{attribute 'call_after_init'}
FUNCTION_BLOCK FB_eVWithinSpec_Test EXTENDS TcUnit.FB_TestSuite
VAR_INPUT
END_VAR
VAR_OUTPUT
END_VAR
VAR
END_VAR

evWithinRangeChecks();

METHOD evWithinRangeChecks
VAR_INPUT
END_VAR
VAR

END_VAR
TEST('evWithinRangeChecks');
	
//Upper limit equal
AssertTrue(
	F_eVWithinSpec(300, 2#0000_0000_0000_0010),
	'Upper limit not inclusive');
//Lower limit equal
AssertTrue(
	F_eVWithinSpec(300, 2#0000_0000_0000_0100),
	'Lower limit not inclusive');
//Out of range
AssertFalse(
	F_eVWithinSpec(300.1, 2#0000_0000_0000_0010),
	'Out of range failed, whatever you did, it broke this really bad.');
//Negative eV
AssertFalse(
	F_eVWithinSpec(-300, 16#FFFF),
	'Working with antimatter? Negative eV should not be acceptable.');
//Upper unallocated range
AssertFalse(
	F_eVWithinSpec(1700, 2#1000_0000_0000_0000),
	'eV range should not evaluate past 1.6keV');
	
TEST_FINISHED();
END_METHOD

END_FUNCTION_BLOCK

(* stored: Version 1.1.0.1, ProductVersion 3.1.4024.0
   POU FB_eVWithinSpec_Test: Id {b622c686-f9dd-0ccb-3e3a-bfb750a08cb0}, SpecialFunc None
   Method evWithinRangeChecks: Id {1d6c611b-6bb7-0728-3075-755617dbc45a} *)
